// TIA Portal project "mixer station working" (V16)
// Vorlageprojekt für das Buch mit Zielsystem S7-1200

(* hardware
DEVICE "S7-1200-Station_1"  S7-1200 Station
   slot 0: "Baugruppenträger_0"  Rack  V1.0
   slot 1: "PLC_1"  CPU 1211C DC/DC/DC  6ES7 211-1AE40-0XB0  V4.1
*)

// ===== PLC "PLC_1"  CPU 1211C DC/DC/DC =====

VAR_GLOBAL   // PLC tag table "Standard-Variablentabelle"
   "start" AT %E0.0 : Bool;
   "emergecy stop" AT %E0.1 : Bool;
   "up sensor" AT %I0.2 : Bool;
   "below sensor" AT %I0.3 : Bool;
   "Tag_1" AT %M0.1 : Bool;
   "Tag_2" AT %M0.2 : Bool;
   "fill pump" AT %Q0.0 : Bool;
   "mixer" AT %Q0.1 : Bool;
   "drain pump" AT %Q0.2 : Bool;
   "Tag_3" AT %M0.4 : Bool;
   "Tag_4" AT %M0.5 : Bool;
   "Tag_5" AT %M0.6 : Bool;
   "Cycle_Count up" AT %QD30 : DInt;
   "Cycle_Count drain" AT %QD34 : DInt;
   "Tag_6" AT %M0.7 : Bool;
   "Tag_7" AT %Q0.3 : Bool;
   "Tag_8" AT %M1.2 : Bool;
   "Tag_9" AT %I0.4 : Bool;
   "Tag_10" AT %M0.3 : Bool;
   "Tag_11" AT %M1.5 : Bool;
END_VAR

// folder: System blocks/Program resources

DATA_BLOCK "IEC_Counter_0_DB"   // DB1
{ S7_Optimized_Access := 'TRUE' }
AUTHOR : Simatic
FAMILY : IEC
NAME : CNTR
VERSION : 1.0
// stored: InstanceOfName IEC_COUNTER
"IEC_COUNTER"
BEGIN
END_DATA_BLOCK

DATA_BLOCK "IEC_Counter_1_DB"   // DB2
{ S7_Optimized_Access := 'TRUE' }
AUTHOR : Simatic
FAMILY : IEC
NAME : CNTR
VERSION : 1.0
// stored: InstanceOfName IEC_COUNTER
"IEC_COUNTER"
BEGIN
END_DATA_BLOCK

DATA_BLOCK "IEC_Timer_0_DB_4"   // DB6
{ S7_Optimized_Access := 'TRUE' }
AUTHOR : Simatic
FAMILY : IEC
NAME : IEC_TMR
VERSION : 1.0
// stored: InstanceOfName IEC_TIMER
"IEC_TIMER"
BEGIN
END_DATA_BLOCK

// folder: (top level)

FUNCTION "MHJ-PLC-Lab-Function-S71200" : Void   // FC9000, SCL
{ S7_Optimized_Access := 'TRUE' }
VERSION : 0.1
   VAR_TEMP
      rdTimeReturn : Int;
      outputTime : DTL;
      SyncVal : Byte;
      forVal : Int;
      forVal_2 : Int;
      Value : Byte;
   END_VAR
   VAR CONSTANT
      CompVal : Byte := 16#34;
      Value_01 : Byte := 16#11;
      Value_01_DW : DWord := 16#A165_D992;
      Value_02_DW : DWord := 16#58BE_4401;
   END_VAR
BEGIN

   #Value:=PEEK(area := 16#82,
        dbNumber := 0,
        byteOffset := 511);
   #Value := #Value + 1;

   POKE(area := 16#82,
        dbNumber := 0,
        byteOffset := 511,
        value := #Value);

   POKE(area:=16#81,
        dbNumber:=0,
        byteOffset:=1016,
        value:=#Value_01_DW);
   POKE(area := 16#81,
        dbNumber := 0,
        byteOffset := 1020,
        value := #Value_02_DW);

   POKE(area := 16#81,
        dbNumber := 0,
        byteOffset := 511,
        value := B#16#00);

   FOR #forVal := 0 TO 120 DO
       FOR #forVal_2:=0 TO 10 DO
           #rdTimeReturn:=RD_SYS_T(#outputTime);
           #rdTimeReturn := WR_SYS_T(#outputTime);
           #rdTimeReturn := RD_SYS_T(#outputTime);
           #rdTimeReturn := WR_SYS_T(#outputTime);
       END_FOR;
       #SyncVal:= PEEK(area := 16#81,
                      dbNumber := 0,
                      byteOffset := 511);
       IF #SyncVal = #CompVal THEN
          GOTO M_1;
       END_IF;
   END_FOR;
   RETURN;

   M_1:
   POKE(area := 16#81,
        dbNumber := 0,
        byteOffset := 511,
        value := B#16#0);
END_FUNCTION

ORGANIZATION_BLOCK "Main"   // OB1, LAD, ProgramCycle
TITLE = "Main Program Sweep (Cycle)"
{ S7_Optimized_Access := 'TRUE' }
VERSION : 0.1
   VAR_INPUT
      Initial_Call : Bool;   // Initial call of this OB
      Remanence : Bool;   // =True, if remanent data are available
   END_VAR
   VAR_TEMP   // added for the SCL form of the ladder/FBD networks
      _w1 : Bool;
   END_VAR
BEGIN

REGION Network 1: Konnektierungsbaustein für PLC-Lab
   // Im Netzwerk 1 wird der Konnektierungsbaustein für PLC-Lab aufgerufen.
   // Dieser Aufruf darf nicht entfernt werden!
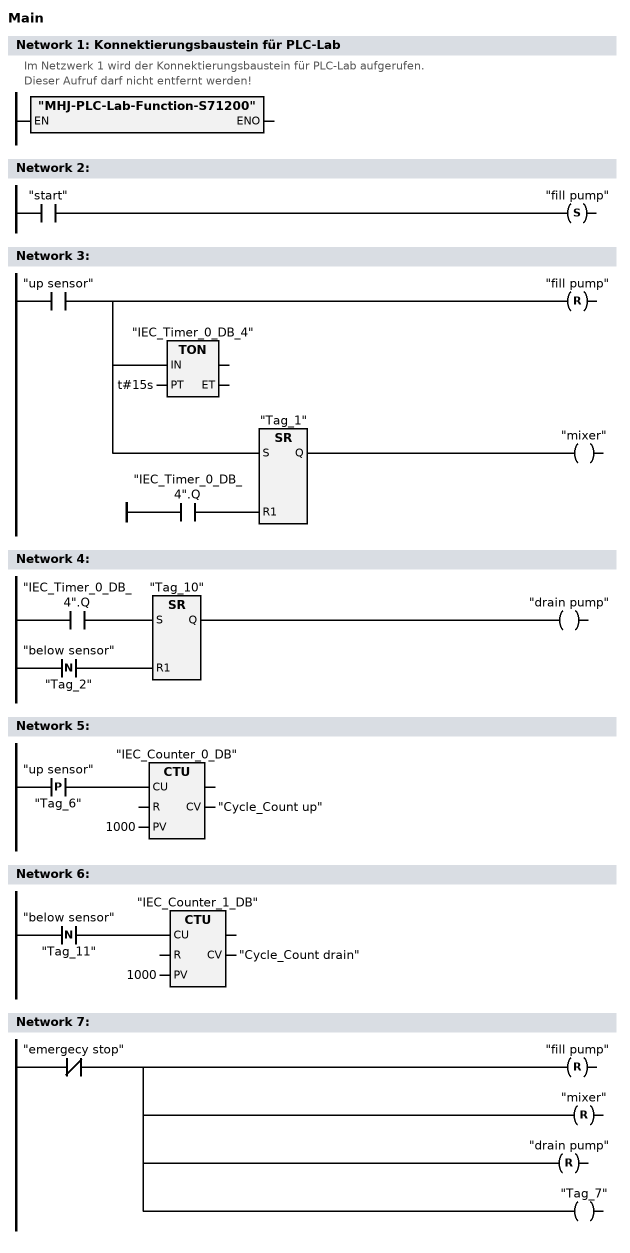
   RUNG wire#powerrail
      "MHJ-PLC-Lab-Function-S71200"()
   END_RUNG
   // the same network as SCL:
   "MHJ-PLC-Lab-Function-S71200"();
END_REGION

REGION Network 2
   RUNG wire#powerrail
      Contact( "start" )
      S_Coil( "fill pump" )
   END_RUNG
   // the same network as SCL:
   IF "start" THEN "fill pump" := TRUE; END_IF;
END_REGION

REGION Network 3
   IF "up sensor" THEN "fill pump" := FALSE; END_IF;
   "IEC_Timer_0_DB_4".TON(IN := "up sensor", PT := t#15s);
   IF "up sensor" THEN
       "Tag_1" := TRUE;   // SR flip-flop
   END_IF;
   IF "IEC_Timer_0_DB_4".Q THEN "Tag_1" := FALSE; END_IF;
   "mixer" := "Tag_1";
END_REGION

REGION Network 4
   RUNG wire#powerrail
      Contact( "IEC_Timer_0_DB_4".Q )
      S_SR(operand := "Tag_10", r1 := wire#w1)
      Coil( "drain pump" )
   END_RUNG
   RUNG wire#powerrail
      N_Contact(operand := "below sensor", bit := "Tag_2")
   END_RUNG wire#w1
   // the same network as SCL:
   #_w1 := NOT "below sensor" AND "Tag_2";   // falling edge of "below sensor"
   "Tag_2" := "below sensor";
   IF "IEC_Timer_0_DB_4".Q THEN
       "Tag_10" := TRUE;   // SR flip-flop
   END_IF;
   IF #_w1 THEN "Tag_10" := FALSE; END_IF;
   "drain pump" := "Tag_10";
END_REGION

REGION Network 5
   #_w1 := "up sensor" AND NOT "Tag_6";   // rising edge of "up sensor"
   "Tag_6" := "up sensor";
   "IEC_Counter_0_DB".CTU(CU := #_w1, PV := 1000, CV => "Cycle_Count up");
END_REGION

REGION Network 6
   #_w1 := NOT "below sensor" AND "Tag_11";   // falling edge of "below sensor"
   "Tag_11" := "below sensor";
   "IEC_Counter_1_DB".CTU(CU := #_w1, PV := 1000, CV => "Cycle_Count drain");
END_REGION

REGION Network 7
   RUNG wire#powerrail
      I_Contact( "emergecy stop" )
      wire#w1
      R_Coil( "fill pump" )
   END_RUNG
   RUNG wire#w1
      R_Coil( "mixer" )
   END_RUNG
   RUNG wire#w1
      R_Coil( "drain pump" )
   END_RUNG
   RUNG wire#w1
      Coil( "Tag_7" )
   END_RUNG
   // the same network as SCL:
   IF NOT "emergecy stop" THEN
       "fill pump" := FALSE;
       "mixer" := FALSE;
       "drain pump" := FALSE;
   END_IF;
   "Tag_7" := NOT "emergecy stop";
END_REGION
END_ORGANIZATION_BLOCK